FUNCTION_BLOCK FB_LightDimmable EXTENDS FB_LightBase IMPLEMENTS I_LightDimmable
VAR
	nBrightness	: USINT := 100;
END_VAR

PROPERTY PUBLIC Brightness : USINT;
GET
Brightness := nBrightness;
END_GET
SET
nBrightness := Brightness;
END_SET
END_PROPERTY

END_FUNCTION_BLOCK

(* stored: Version 1.1.0.1, ProductVersion 3.1.4024.12
   POU FB_LightDimmable: Id {f14caa0a-722a-4bf1-a6f2-9567e3a30e6c}, SpecialFunc None
   Property Brightness: Id {66812941-e28d-4f85-abaf-bc91cf97780e}
   Get Get: Id {ff93fac2-27a7-447a-8b08-a19ebb311b66}
   Set Set: Id {332e252e-81df-40d2-af75-1dcc264f4c22} *)
